Omron CX-Programmer project NewProject (CX-Programmer 9.61)

# PLC NewPLC1: CP1E N30

## Global symbols (name address type ; comment)
0.00 BOOL  ; I_StartButonu
0.01 BOOL  ; I_UstMotorAsagiButon
0.02 BOOL  ; I_OrtaMotorIleriButon
0.03 BOOL  ; I_AltMotorYukariButon
0.04 BOOL  ; I_AcilStopButonu
0.05 BOOL  ; I_BasincSartel
0.06 BOOL  ; I_KapiSw
0.07 BOOL  ; I_StartButon2
100.00 BOOL  ; O_UstMotorAsagiValfi
100.01 BOOL  ; O_OrtaMotorIleriValfi
100.02 BOOL  ; O_AltMotorYukariValfi
100.03 BOOL  ; O_TablaHareketValfi
100.04 BOOL  ; O_SurucuStart
D0 CHANNEL  ; timergerii
T000 BOOL  ; PistonlarIleriTimer
T001 BOOL  ; TablarIleriTimer
T002 BOOL  ; SurucuDonusOkTimer
T012 BOOL  ; CiftElTimer
T013 BOOL  ; CiftElTimer1
W0.00 BOOL  ; SistemOk
W0.01 BOOL  ; SistemStart
W0.02 BOOL  ; dongusonu
W1.00 BOOL  ; IlkStartBasildi
W1.01 BOOL  ; IkinciStartBasildi
W3.00 BOOL  ; CiftElCalismaIptal
W3.01 BOOL  ; CiftElCalismaIptal1

## Program NewProgram1 (cyclic task 0)

### Section Section1

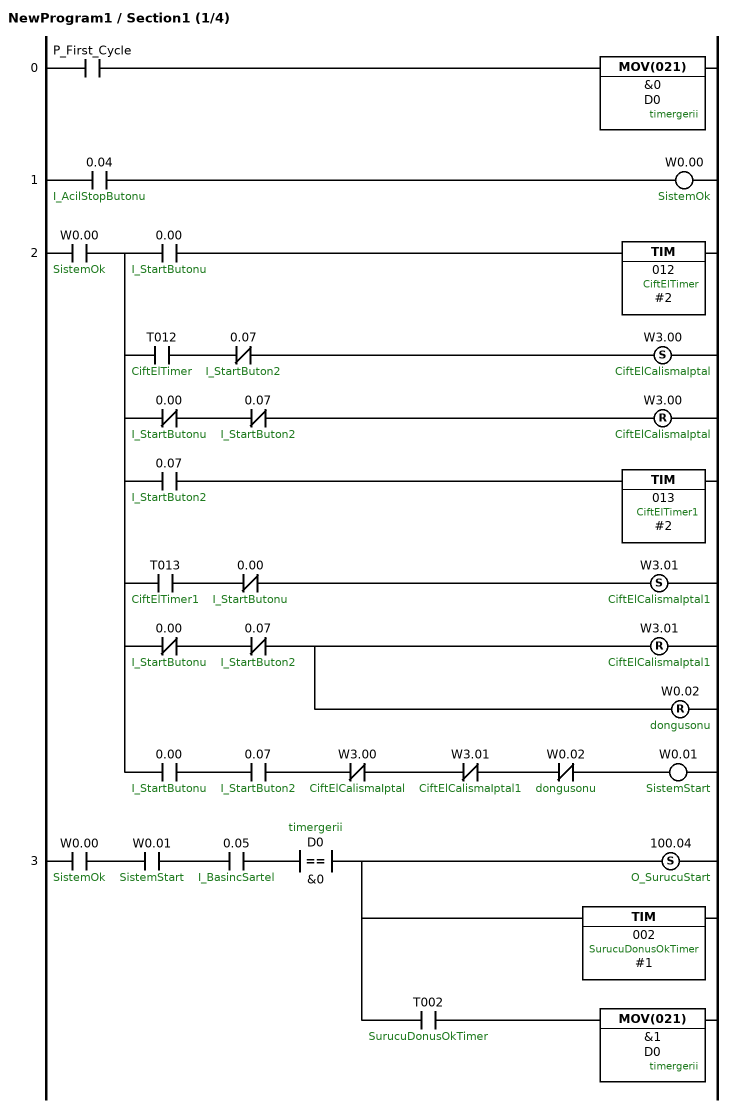
; rung 0
LD P_First_Cycle
MOV(021) &0 D0  ; timergerii
; rung 1
LD 0.04  ; I_AcilStopButonu
OUT W0.00  ; SistemOk
; rung 2
LD W0.00  ; SistemOk
OUT TR0
AND 0.00  ; I_StartButonu
TIM 012 #2  ; CiftElTimer
LD TR0
AND T012  ; CiftElTimer
ANDNOT 0.07  ; I_StartButon2
SET W3.00  ; CiftElCalismaIptal
LD TR0
ANDNOT 0.00  ; I_StartButonu
ANDNOT 0.07  ; I_StartButon2
RSET W3.00  ; CiftElCalismaIptal
LD TR0
AND 0.07  ; I_StartButon2
TIM 013 #2  ; CiftElTimer1
LD TR0
AND T013  ; CiftElTimer1
ANDNOT 0.00  ; I_StartButonu
SET W3.01  ; CiftElCalismaIptal1
LD TR0
ANDNOT 0.00  ; I_StartButonu
ANDNOT 0.07  ; I_StartButon2
RSET W3.01  ; CiftElCalismaIptal1
RSET W0.02  ; dongusonu
LD TR0
AND 0.00  ; I_StartButonu
AND 0.07  ; I_StartButon2
ANDNOT W3.00  ; CiftElCalismaIptal
ANDNOT W3.01  ; CiftElCalismaIptal1
ANDNOT W0.02  ; dongusonu
OUT W0.01  ; SistemStart
; rung 3
LD W0.00  ; SistemOk
AND W0.01  ; SistemStart
AND 0.05  ; I_BasincSartel
AND=(300) D0 &0  ; timergerii
SET 100.04  ; O_SurucuStart
TIM 002 #1  ; SurucuDonusOkTimer
AND T002  ; SurucuDonusOkTimer
MOV(021) &1 D0  ; timergerii

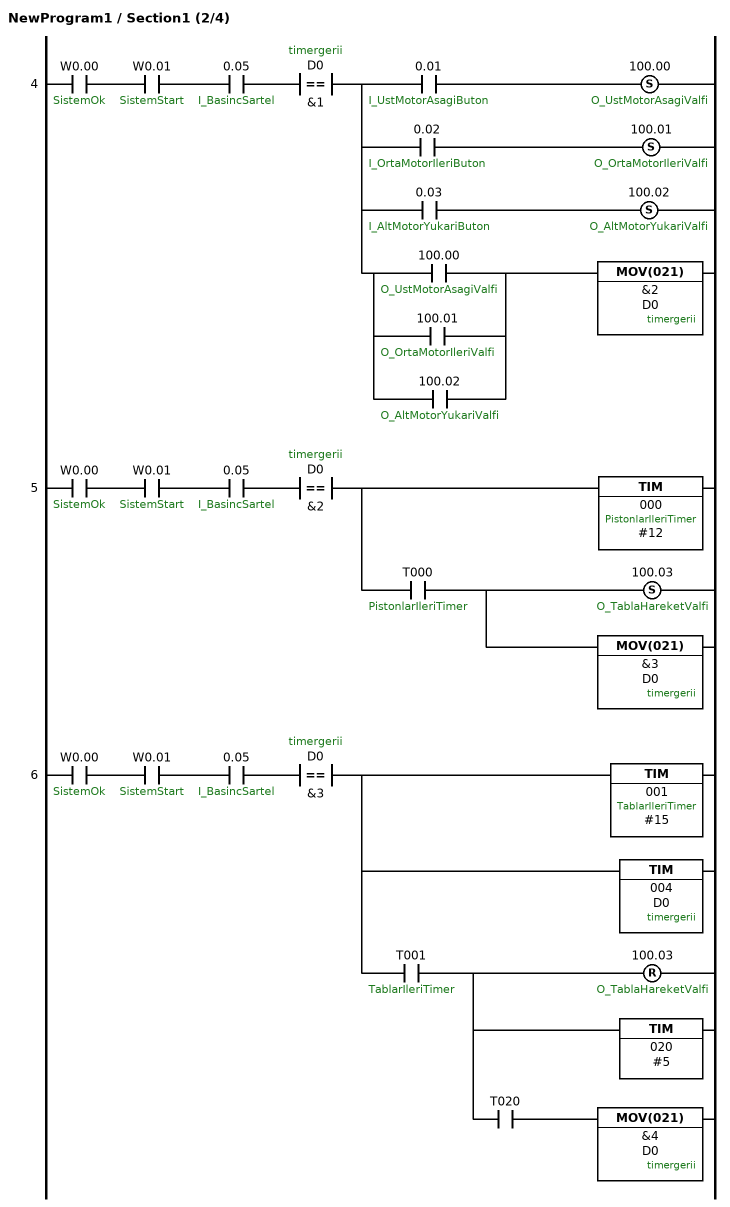
; rung 4
LD W0.00  ; SistemOk
AND W0.01  ; SistemStart
AND 0.05  ; I_BasincSartel
AND=(300) D0 &1  ; timergerii
OUT TR0
AND 0.01  ; I_UstMotorAsagiButon
SET 100.00  ; O_UstMotorAsagiValfi
LD TR0
AND 0.02  ; I_OrtaMotorIleriButon
SET 100.01  ; O_OrtaMotorIleriValfi
LD TR0
AND 0.03  ; I_AltMotorYukariButon
SET 100.02  ; O_AltMotorYukariValfi
LD TR0
LD 100.00  ; O_UstMotorAsagiValfi
OR 100.01  ; O_OrtaMotorIleriValfi
OR 100.02  ; O_AltMotorYukariValfi
ANDLD
MOV(021) &2 D0  ; timergerii
; rung 5
LD W0.00  ; SistemOk
AND W0.01  ; SistemStart
AND 0.05  ; I_BasincSartel
AND=(300) D0 &2  ; timergerii
TIM 000 #12  ; PistonlarIleriTimer
AND T000  ; PistonlarIleriTimer
SET 100.03  ; O_TablaHareketValfi
MOV(021) &3 D0  ; timergerii
; rung 6
LD W0.00  ; SistemOk
AND W0.01  ; SistemStart
AND 0.05  ; I_BasincSartel
AND=(300) D0 &3  ; timergerii
TIM 001 #15  ; TablarIleriTimer
TIM 004 D0  ; timergerii
AND T001  ; TablarIleriTimer
RSET 100.03  ; O_TablaHareketValfi
TIM 020 #5
AND T020
MOV(021) &4 D0  ; timergerii

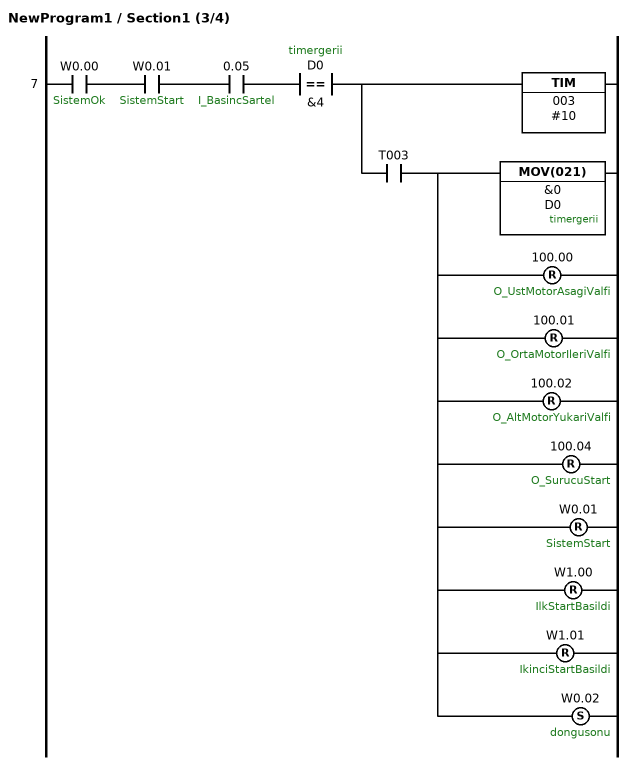
; rung 7
LD W0.00  ; SistemOk
AND W0.01  ; SistemStart
AND 0.05  ; I_BasincSartel
AND=(300) D0 &4  ; timergerii
TIM 003 #10
AND T003
MOV(021) &0 D0  ; timergerii
RSET 100.00  ; O_UstMotorAsagiValfi
RSET 100.01  ; O_OrtaMotorIleriValfi
RSET 100.02  ; O_AltMotorYukariValfi
RSET 100.04  ; O_SurucuStart
RSET W0.01  ; SistemStart
RSET W1.00  ; IlkStartBasildi
RSET W1.01  ; IkinciStartBasildi
SET W0.02  ; dongusonu

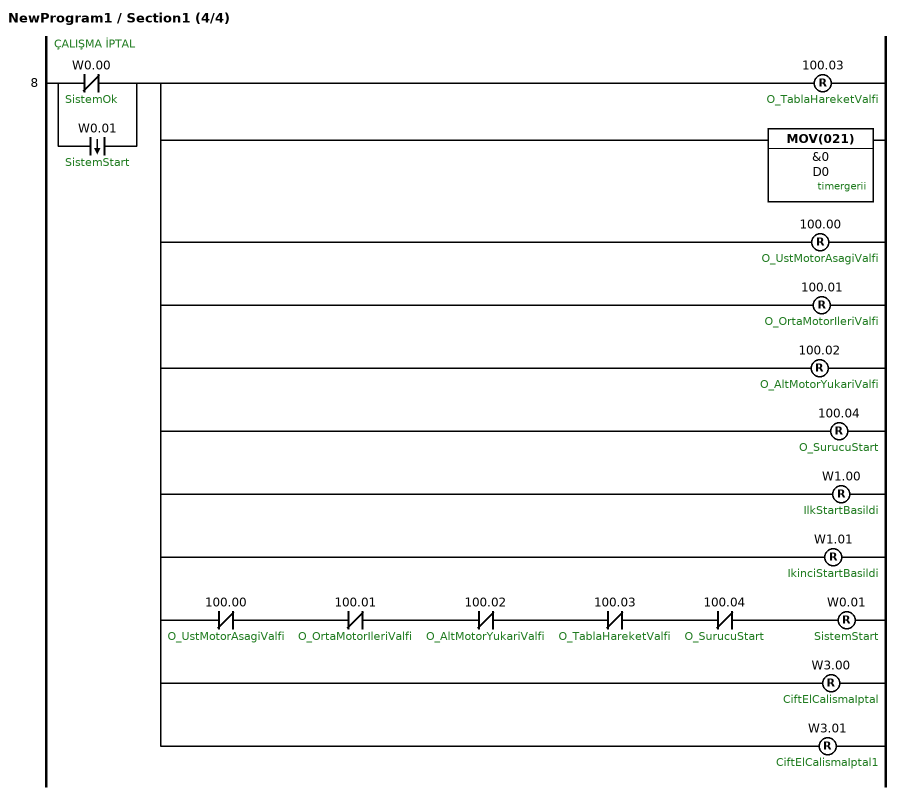
; rung 8: ÇALIŞMA İPTAL
LDNOT W0.00  ; SistemOk
%OR W0.01  ; SistemStart
OUT TR0
RSET 100.03  ; O_TablaHareketValfi
MOV(021) &0 D0  ; timergerii
RSET 100.00  ; O_UstMotorAsagiValfi
RSET 100.01  ; O_OrtaMotorIleriValfi
RSET 100.02  ; O_AltMotorYukariValfi
RSET 100.04  ; O_SurucuStart
RSET W1.00  ; IlkStartBasildi
RSET W1.01  ; IkinciStartBasildi
ANDNOT 100.00  ; O_UstMotorAsagiValfi
ANDNOT 100.01  ; O_OrtaMotorIleriValfi
ANDNOT 100.02  ; O_AltMotorYukariValfi
ANDNOT 100.03  ; O_TablaHareketValfi
ANDNOT 100.04  ; O_SurucuStart
RSET W0.01  ; SistemStart
LD TR0
RSET W3.00  ; CiftElCalismaIptal
RSET W3.01  ; CiftElCalismaIptal1

### Section END
; rung 0
END(001)